Staubli VAL3: onRun.pgx

public program onRun(string& x_sItem[])
  local num l_nValue
  local num l_nValue1
  local num l_nVelocity
begin
  //
  // Done, when you execute it
  //
  ////  call findValue(x_sItem,l_nValue)
  ////  aioSet(io:movePulse,l_nValue)
  ////  io:move=true
  ////  delay(0.5)
  ////  io:move=false
  ////  wait(io:atPosition==true or isKeyPressed(255))
  if aioGet(MbAI_bBackHome)!=1
    popUpMsg("7轴未回零位，请先执行回零位操作")
    return
  endIf
  aioSet(MbAO_b7Axis,1)
  aioSet(MbAO_aMoveDis,0)
  aioSet(MbAO_bMoveToPos,0)
  bAxisRun=true
//  aioSet(MbAI_bAxis7Reac,0)
  delay(0.5)
  call findValue(x_sItem,l_nValue,l_nValue1)
  call getVelocity(x_sItem,l_nVelocity)
  l_nVelocity=l_nVelocity*1000/60
  aioSet(MbAO_aMovePosL,l_nValue)
  aioSet(MbAO_aMovePosH,l_nValue1)
  aioSet(MbAO_aVelocity,l_nVelocity)
  aioSet(MbAO_bMoveToPos,1)
  delay(0.5)
  wait(aioGet(MbAI_bAxis7Reac)==0)
  wait(aioGet(MbAI_bAxis7Reac)==1 or isKeyPressed(255))
  if isKeyPressed(255)
    //if !cycleStatus:bCycle and !cycleStatus:bSimulation
      if aioGet(MbAO_bStopMotor)==1
        aioSet(MbAO_bStopMotor,0)
        delay(0.2)
        aioSet(MbAO_bStopMotor,1)
        delay(0.2)
      else
        aioSet(MbAO_bStopMotor,1)
        delay(0.4)
        aioSet(MbAO_bStopMotor,0)
      endIf
    //endIf
  endIf
  aioSet(MbAO_bMoveToPos,0)
  aioSet(MbAO_b7Axis,0)
  logMsg("1")
  // aioSet(io:MbAI_bAxis7Reac,0)
  bAxisRun=false
end
